// TIA Portal V15 export
// export: Created 2018-05-29T12:25:38.1552518Z, ExportSetting WithDefaults, DisplayName Totally Integrated Automation Portal, DisplayVersion V15, DisplayName STEP 7 Professional, DisplayVersion V15, DisplayName WinCC Professional, DisplayVersion V15, DisplayName TIA Portal Openness, DisplayVersion V15
FUNCTION "EM_Instance_14_fc" : Void   // FC1, STL
TITLE = _fc
{ S7_Optimized_Access := 'TRUE' }
VERSION : 0.1
// test
// stored: AutoNumber true, UDAEnableTagReadback false
BEGIN

NETWORK
TITLE = Main
// comment:


// Call the EM FB with the corresponding DB instance
      CALL  "EM_I_OUT", "EM_Instance_14"
      ( sampletime       := ,
        em_id            := #"39",
        Request          := ,
        Command          := ,
        Pressure_SP      := ,
        Pump_RUN         := #"M106.QNOFF2",
        Pump_QERR        := #"M106.QERR",
        Pump_EERR        := #"M106.QERR_EXT",
        FS01_PV          := #"LS002.QON",
        PIC01_PV         := #"FIC101.PV",
        PIC01_ERR        := #"FIC101.QERR",
        LT01_PV          := #"LT201.QfVal",
        LT01_AHH         := #"LT201.LIM_Qb01",
        LT01_AH          := #"LT201.LIM_Qb02",
        LT01_AL          := #"LT201.LIM_Qb03",
        LT01_ALL         := #"LT201.LIM_Qb04",
        LT01_ERR         := #"LT201.QERR",
        XV_Bottom_OPN    := #"XV004.QOPEN",
        XV_Bottom_CLS    := #"XV004.QCLOSE",
        XV_Bottom_MERR   := #"XV004.QMON_ERR",
        BV_Bottom_OPN    := ,
        BV_Bottom_CLS    := ,
        BV_Bottom_MERR   := ,
        BV_Tran_M04_OPN  := ,
        BV_Tran_M04_CLS  := ,
        BV_Tran_M04_MERR := ,
        steptime_s       := ,
        steptime_m       := ,
        steptime_h       := ,
        first_scan       := ,
        last_scan        := ,
        error_index_db   := ,
        Owner            := ,
        Status           := ,
        CM_error         := ,
        CM_error_no      := ,
        q_bACTVIE        := ,
        Level            := ,
        Pressure         := ,
        Pump_ON          := #"M106.L_ON",
        Pump_AUT         := #"M106.L_AUT",
        PIC01_EXT        := #"FIC101.L_REMOTE",
        PIC01_SP         := #"FIC101.HMI_SP_INT",
        PIC01_AUT        := #"FIC101.L_AUT",
        PIC01_VAL_OUT    := #"FIC101.HMI_MAN",
        PIC01_SET_SP     := #"FIC101.Set_SP",
        PIC01_SET_OUT    := #"FIC101.Set_Output",
        XV_Bottom_CMD    := #"XV004.AUT_OP",
        BV_Bottom_CMD    := ,
        BV_Tran_M04_CMD  := 
      );
END_FUNCTION
